Staubli VAL3: Action.pgx

public program Action(num& x_nAction[] (dimensions=2), bool x_bMoveId, num x_nMoveID)
  local bool l_bFirst
  local bool l_bInput
  local bool l_bNull
  local num l_nLast
  local num l_nNum
begin
  //延时是否需要停止等待？
  //




  //一共是每个点上最多12个IO


  //如果都为空，则直接跳出
  l_bNull=false
  for l_nNum=0 to 11
    l_bNull=x_nAction[l_nNum,0]!=0 or x_nAction[l_nNum,1]!=0 or l_bNull
  endFor
  if !l_bNull
    return
  endIf




  //通过MOVEID来实现
  for l_nNum=0 to 11

    //如果后面的都是0则退出
    l_bNull=false
    for l_nLast=l_nNum to 11
      l_bNull=x_nAction[l_nLast,0]!=0 or x_nAction[l_nLast,1]!=0 or l_bNull
    endFor
    if !l_bNull
      return
    endIf


    //通过MOVEID来实现
    if x_bMoveId
      call IsInput(x_nAction[l_nNum,0],l_bInput)
      //如果有等待信号，直接退出
      if l_bInput
        return
      else
        wait(getMoveId()>x_nMoveID+0.8)
        call IOvalue(x_nAction[l_nNum,0],x_nAction[l_nNum,1])
      endIf





     //
    else

      //跟在运动指令后面
      call IsInput(x_nAction[l_nNum,0],l_bInput)
      //如果有等待信号 则运行
      if l_bInput
        l_bFirst=true

      endIf

      if l_bFirst
        //如果不是收弧时间


        if x_nAction[l_nNum,0]!=166 and l_bInput
          if x_nMoveID==-2
            waitEndMove()
          else
            if x_nMoveID>=0
              wait(getMoveId()>x_nMoveID+0.8)
            endIf
          endIf
        endIf
      endIf

      call IOvalue(x_nAction[l_nNum,0],x_nAction[l_nNum,1])


      if x_nAction[l_nNum,0]==166
        //  logMsg(toString(".3",x_nAction[l_nNum,1]))
        logMsg(toString(".3",clock())+"  "+toString(".3",getMoveId()))
      endIf


    endIf


    //把数字量输出
    call Digtal2Analog()

  endFor


end
